	                *)
	                #PO_INVT.CTW.%B1 := 1;
	                IF "Zona".Z[#K_Zona].Gen.Reset AND ("Motore".M[#K_MotoreInt].Dati.MotoreFermo OR "Motore".M[#K_MotoreInt].In.DriverFault) THEN
	                    #PO_INVT.CTW.%B0 := 7;
	                ELSIF "Motore".M[#K_MotoreInt].Out.CmdPosMotore THEN
	                    #PO_INVT.CTW.%B0 := 1;
	                ELSIF "Motore".M[#K_MotoreInt].Out.CmdNegMotore THEN
	                    #PO_INVT.CTW.%B0 := 2;
	                ELSE
	                    #PO_INVT.CTW.%B0 := 6;
	                END_IF;
	                #PO_INVT.CTW.%X15 := NOT #PI_INVT.STW.%X15;
	                #PO_INVT.Speed := DINT_TO_INT(TRUNC("Motore".M[#K_MotoreInt].Out.VelAss / DINT_TO_REAL("Motore".M[#K_MotoreInt].Prm.C.VelMax) * 10000.0));
	                REGION ScritturaParametri
	                    IF #PI_INVT.PKW01 <> 0 THEN
	                        IF "Motore".M[#K_MotoreInt].Dati.PrmSend THEN
	                            "Motore".M[#K_MotoreInt].Dati.IdPrm += 1;
	                            IF "Motore".M[#K_MotoreInt].Dati.IdPrm > 1 THEN
	                                "Motore".M[#K_MotoreInt].Dati.IdPrm := 0;
	                            END_IF;
	                            "Motore".M[#K_MotoreInt].Dati.PrmSend := false;
	                        END_IF;
	                    ELSE
	                        "Motore".M[#K_MotoreInt].Dati.PrmSend := true;
	                        CASE "Motore".M[#K_MotoreInt].Dati.IdPrm OF
	                            0:  //Acc
	                                #PO_INVT.PKW01 := 4;
	                                #PO_INVT.PKW02 := 11;
	                                #PO_INVT.PKW04 := DINT_TO_WORD(TRUNC(DINT_TO_REAL("Motore".M[#K_MotoreInt].Prm.C.VelMax) / DINT_TO_REAL("Motore".M[#K_MotoreInt].Prm.DecEmergenza) * 3.0));
	                            1:  //Dec
	                                #PO_INVT.PKW01 := 4;
	                                #PO_INVT.PKW02 := 12;
	                                #PO_INVT.PKW04 := DINT_TO_WORD(TRUNC(DINT_TO_REAL("Motore".M[#K_MotoreInt].Prm.C.VelMax) / DINT_TO_REAL("Motore".M[#K_MotoreInt].Prm.DecEmergenza) * 3.0));
	                            ELSE
	                                "Motore".M[#K_MotoreInt].Dati.PrmSend := false;
	                                "Motore".M[#K_MotoreInt].Dati.IdPrm := 0;
	                        END_CASE;
	                    END_IF;
	                END_REGION
	                "Motore".M[#K_MotoreInt].Dati.RetVal_SCR_Inv := DPWR_DAT(LADDR := "Motore".M[#K_MotoreInt].HW.HWIO_Inverter, RECORD := #PO_INVT);
	                "Motore".M[#K_MotoreInt].HMI.CTW1 := #PO_INVT.CTW;
	            END_REGION
	        9:
	            REGION Nidec
	                (*
	                BIT 00: Drive Enable
	                BIT 01: Run Forward
	                BIT 02: Jog Forward
	                BIT 03: Run Reverse
	                BIT 04: Forward/Reverse
	                BIT 05: Run
	                BIT 06: Not Stop
	                BIT 07: Auto / manual
	                BIT 08: Analog / Preset reference
	                BIT 09: Jog Reverse
	                BIT 10: Not used
	                BIT 11: Not used
	                BIT 12: Trip drive
	                BIT 13: Reset drive
	                BIT 14: Watchdog
	                *)
	                #PO_Nidec.CTW.%X7 := true;
	                #PO_Nidec.CTW.%X0 := #PO_Nidec.CTW.%X6 := #PI_Nidec.STW.%X0 AND "Zona".Z[#K_ZonaInt].Out.CentralinaOk;
	                //#PO_Nidec.CTW.%X1 := "Motor".M[#MotorNumber].o.CmdFWD OR "Motor".M[#MotorNumber].o.CmdBKW;
	                //#PO_Nidec.CTW.%X3 := "Motor".M[#MotorNumber].o.CmdBKW;
	                #PO_Nidec.CTW.%X5 := "Motore".M[#K_MotoreInt].Out.CmdPosMotore OR "Motore".M[#K_MotoreInt].Out.CmdNegMotore;
	                #PO_Nidec.CTW.%X4 := "Motore".M[#K_MotoreInt].Out.CmdNegMotore;
	                #PO_Nidec.CTW.%X13 := "Zona".Z[#K_Zona].Gen.Reset AND "Motore".M[#K_MotoreInt].In.DriverFault;
	                #PO_Nidec.Speed := TRUNC("Motore".M[#K_MotoreInt].Out.VelAss / DINT_TO_REAL("Motore".M[#K_MotoreInt].Prm.C.VelMax) * 10000.0);
	                #PO_Nidec.RampAcc := TRUNC(DINT_TO_REAL("Motore".M[#K_MotoreInt].Prm.C.VelMax) / DINT_TO_REAL("Motore".M[#K_MotoreInt].Dati.AccRichPerc) * 3.0);
	                #PO_Nidec.RampDec := TRUNC(DINT_TO_REAL("Motore".M[#K_MotoreInt].Prm.C.VelMax) / DINT_TO_REAL("Motore".M[#K_MotoreInt].Dati.DecReqEmergInLavo) * 3.0);
	                "Motore".M[#K_MotoreInt].HMI.CTW1 := #PO_Nidec.CTW;
	                //VariantPut(SRC := #PO_Nidec, DST := #PO_Inv);
	            END_REGION
	            ;
	    END_CASE;
	END_REGION ;
	REGION Update
	    IF "Motore".M[#K_MotoreInt].HMI.UpdParam THEN
	        "Motore".M[#K_MotoreInt].HMI.UpdParam := FALSE;
	        "Motore".M[#K_MotoreInt].Out.UpdParam := true;
	    ELSE
	        IF "Motore".M[#K_MotoreInt].Out.UpdParam THEN
	            "Motore".M[#K_MotoreInt].HMI.FBGestione := 100 + "Motore".M[#K_MotoreInt].HW.TipoCollInverter;
	            CASE "Motore".M[#K_MotoreInt].HW.TipoEncoder OF
	                1: // ENCODER SICK
	                    "Motore".M[#K_MotoreInt].Dati.Encoder.RicircoloEncoder := 1073741824;
	                    "Motore".M[#K_MotoreInt].Dati.Encoder.MezzoRicircoloEncoder := "Motore".M[#K_MotoreInt].Dati.Encoder.RicircoloEncoder / 2;
	                    "Motore".M[#K_MotoreInt].Prm.Enc.ImpRev := 262144.0;
	                10, 11: // ENCODER T+R
	                    "Motore".M[#K_MotoreInt].Dati.Encoder.RicircoloEncoder := 16#0200_0000;
	                    "Motore".M[#K_MotoreInt].Dati.Encoder.MezzoRicircoloEncoder := "Motore".M[#K_MotoreInt].Dati.Encoder.RicircoloEncoder / 2;
	                    "Motore".M[#K_MotoreInt].Prm.Enc.ImpRev := 8192.0;
	            END_CASE;
	        END_IF;
	        "Motore".M[#K_MotoreInt].Out.UpdParam := false;
	    END_IF;
	    IF "Motore".M[#K_MotoreInt].Out.UpdParam THEN
	        "Motore".M[#K_MotoreInt].In.Positioning := false;
	        "Motore".M[#K_MotoreInt].In.PosRelativo := false;
	        "Motore".M[#K_MotoreInt].In.CambioVelDaPunto := false;
	        "Motore".M[#K_MotoreInt].In.CmdPosRich := false;
	        "Motore".M[#K_MotoreInt].In.CmdNegRich := false;
	        "Motore".M[#K_MotoreInt].In.MotoreRun := false;
	        "Motore".M[#K_MotoreInt].In.AttivaLimVarPos := false;
	        "Motore".M[#K_MotoreInt].In.AttivaLimVarNeg := false;
	        "Motore".M[#K_MotoreInt].In.Premagnetizza := false;
	        "Motore".M[#K_MotoreInt].In.PremagnetizzaPos := false;
	        "Motore".M[#K_MotoreInt].In.PremagnetizzaNeg := false;
	        "Motore".M[#K_MotoreInt].In.ForzaEndLessPos := false;
	        "Motore".M[#K_MotoreInt].In.ForzaEndLessNeg := false;
	        "Motore".M[#K_MotoreInt].In.ForzaEndLessBreve := false;
	        "Motore".M[#K_MotoreInt].In.SezAperto := false;
	        "Motore".M[#K_MotoreInt].In.DriverFault := false;
	        "Motore".M[#K_MotoreInt].In.DriverWarning := false;
	        "Motore".M[#K_MotoreInt].In.NoComunInv := false;
	        "Motore".M[#K_MotoreInt].In.NoComunEnc := false;
	        "Motore".M[#K_MotoreInt].In.TerVentolaOff := false;
	        "Motore".M[#K_MotoreInt].In.CinghiaRotta := false;
	        "Motore".M[#K_MotoreInt].In.SensAzz := false;
	        "Motore".M[#K_MotoreInt].In.SpinaSicNoInPos := false;
	        "Motore".M[#K_MotoreInt].In.ConsMovimentoPos := true;
	        "Motore".M[#K_MotoreInt].In.ConsMovimentoNeg := true;
	        "Motore".M[#K_MotoreInt].In.AnticadutaOFF := false;
	        "Motore".M[#K_MotoreInt].In.AnticadutaON := false;
	        "Motore".M[#K_MotoreInt].In.PercentualeRichiesta := 100;
	        "Motore".M[#K_MotoreInt].Out.CmdPosMotore := false;
	        "Motore".M[#K_MotoreInt].Out.CmdNegMotore := false;
	        "Motore".M[#K_MotoreInt].Out.CmdAnticaduta := false;
	        "Motore".M[#K_MotoreInt].Out.Paw := 0;
	        "Motore".M[#K_MotoreInt].Out.VelEncoder := 0;
	        "Motore".M[#K_MotoreInt].Prm.ByPassAnticaduta := false;
	        "Motore".M[#K_MotoreInt].Prm.AnticadutaPresente := false;
	        "Motore".M[#K_MotoreInt].Prm.PremaNoFreno := false;
	        "Motore".M[#K_MotoreInt].Prm.EscludiFunzPos := false;
	        "Motore".M[#K_MotoreInt].Prm.CambioDirNoFreno := false;
	        "Motore".M[#K_MotoreInt].Prm.CalcTempoRimanente := false;
	        "Motore".M[#K_MotoreInt].Prm.FrenoPresente := false;
	        "Motore".M[#K_MotoreInt].Prm.DisabCicloAutoAllarme := false;
	        "Motore".M[#K_MotoreInt].Prm.DisabCicloManuAllarme := false;
	        "Motore".M[#K_MotoreInt].HMI.Setup := false;
	        "Motore".M[#K_MotoreInt].HMI.ManMov := false;
	        "Motore".M[#K_MotoreInt].HMI.Param.Read := false;
	        "Motore".M[#K_MotoreInt].HMI.Param.Write := false;
	        "Motore".M[#K_MotoreInt].HMI.Param.Save := false;
	        "Motore".M[#K_MotoreInt].HMI.Param.FactoryInit := false;
	        "Motore".M[#K_MotoreInt].HMI.Param.Init_Motor := false;
	        "Motore".M[#K_MotoreInt].HMI.FBGestione := 100 + "Motore".M[#K_MotoreInt].HW.TipoCollInverter;
	        CASE "Motore".M[#K_MotoreInt].HW.TipoEncoder OF
	            1: // ENCODER SICK
	                "Motore".M[#K_MotoreInt].Dati.Encoder.RicircoloEncoder := 1073741824;
	                "Motore".M[#K_MotoreInt].Dati.Encoder.MezzoRicircoloEncoder := "Motore".M[#K_MotoreInt].Dati.Encoder.RicircoloEncoder / 2;
	                "Motore".M[#K_MotoreInt].Prm.Enc.ImpRev := 262144.0;
	            10, 11: // ENCODER T+R
	                "Motore".M[#K_MotoreInt].Dati.Encoder.RicircoloEncoder := 16#0200_0000;
	                "Motore".M[#K_MotoreInt].Dati.Encoder.MezzoRicircoloEncoder := "Motore".M[#K_MotoreInt].Dati.Encoder.RicircoloEncoder / 2;
	                "Motore".M[#K_MotoreInt].Prm.Enc.ImpRev := 8192.0;
	        END_CASE;
	        REGION CalcoloSviluppoEncoder
	            CASE "Motore".M[#K_MotoreInt].Prm.Enc.Mounting OF
	                1:
	                    // Albero Lento
	                    "Motore".M[#K_MotoreInt].Prm.C.SpazioGiroEncoder := UDINT_TO_REAL("Motore".M[#K_MotoreInt].Prm.Mech.FeedConstant);
	                2:
	                    // Albero Veloce
	                    "Motore".M[#K_MotoreInt].Prm.C.SpazioGiroEncoder := UDINT_TO_REAL("Motore".M[#K_MotoreInt].Prm.Mech.FeedConstant * "Motore".M[#K_MotoreInt].Prm.Mech.GearIn) / DINT_TO_REAL("Motore".M[#K_MotoreInt].Prm.Mech.GearOut);
	                ELSE
	                    "Motore".M[#K_MotoreInt].Prm.C.SpazioGiroEncoder := UDINT_TO_REAL("Motore".M[#K_MotoreInt].Prm.Enc.FeedConstant);
	            END_CASE;
	        END_REGION
	        "Motore".M[#K_MotoreInt].Prm.C.VelMax := TRUNC(UDINT_TO_REAL("Motore".M[#K_MotoreInt].Prm.Mech.FeedConstant) * (DINT_TO_REAL("Motore".M[#K_MotoreInt].Prm.Mech.GearIn) / DINT_TO_REAL("Motore".M[#K_MotoreInt].Prm.Mech.GearOut)) * DINT_TO_REAL("Motore".M[#K_MotoreInt].Prm.Mech.RPMMaxRef) / 60.0);
	        CASE "Motore".M[#K_MotoreInt].HMI.ModoInizializza OF
	            1:
	                "Motore".M[#K_MotoreInt].Prm.TMinVCost := 200;
	                "Motore".M[#K_MotoreInt].Prm.TCambioDir := 200;
	                IF "Motore".M[#K_MotoreInt].HW.TipoCollInverter <> 0 THEN
	                    "Motore".M[#K_MotoreInt].Prm.VelPrema := 1;
	                ELSE
	                    "Motore".M[#K_MotoreInt].Prm.VelPrema := "Motore".M[#K_MotoreInt].Prm.C.VelMax / 100;
	                END_IF;
	                "Motore".M[#K_MotoreInt].Prm.VelBassa := "Motore".M[#K_MotoreInt].Prm.C.VelMax / 10;
	                "Motore".M[#K_MotoreInt].Prm.VelSgancioFrenoPos := "Motore".M[#K_MotoreInt].Prm.C.VelMax / 50;
	                "Motore".M[#K_MotoreInt].Prm.VelSgancioFrenoNeg := "Motore".M[#K_MotoreInt].Prm.C.VelMax / 50;
	                "Motore".M[#K_MotoreInt].Prm.SpazioArrestoPos := "Motore".M[#K_MotoreInt].Prm.C.VelMax / 500;
	                "Motore".M[#K_MotoreInt].Prm.SpazioArrestoNeg := "Motore".M[#K_MotoreInt].Prm.C.VelMax / 500;
	                "Motore".M[#K_MotoreInt].Prm.Precisione := MAX(IN1 := "Motore".M[#K_MotoreInt].Prm.SpazioArrestoPos, IN2 := "Motore".M[#K_MotoreInt].Prm.SpazioArrestoNeg) * 2;
	                "Motore".M[#K_MotoreInt].Prm.Inerzia := "Motore".M[#K_MotoreInt].Prm.Precisione + 2000;
	                "Motore".M[#K_MotoreInt].Prm.DecFinale := "Motore".M[#K_MotoreInt].Prm.C.VelMax * 2;
	                "Motore".M[#K_MotoreInt].Prm.DecEmergenza := "Motore".M[#K_MotoreInt].Prm.C.VelMax * 3;
	                "Motore".M[#K_MotoreInt].In.Acc := "Motore".M[#K_MotoreInt].Prm.C.VelMax * 2;
	                "Motore".M[#K_MotoreInt].In.Dec := "Motore".M[#K_MotoreInt].Prm.C.VelMax * 2;
	                "Motore".M[#K_MotoreInt].Prm.VelMan := "Motore".M[#K_MotoreInt].Prm.C.VelMax / 4;
	                "Motore".M[#K_MotoreInt].Prm.VelJog := "Motore".M[#K_MotoreInt].Prm.C.VelMax / 10;
	                "Motore".M[#K_MotoreInt].Prm.ValMaxRef := 27648;
	            2:
	                "Motore".M[#K_MotoreInt].Prm.TMinVCost := 200;
	                "Motore".M[#K_MotoreInt].Prm.TCambioDir := 200;
	                IF "Motore".M[#K_MotoreInt].HW.TipoCollInverter <> 0 THEN
	                    "Motore".M[#K_MotoreInt].Prm.VelPrema := 1;
	                ELSE
	                    "Motore".M[#K_MotoreInt].Prm.VelPrema := "Motore".M[#K_MotoreInt].Prm.C.VelMax / 100;
	                END_IF;
	                "Motore".M[#K_MotoreInt].Prm.VelBassa := "Motore".M[#K_MotoreInt].Prm.C.VelMax / 10;
	                "Motore".M[#K_MotoreInt].Prm.VelSgancioFrenoPos := "Motore".M[#K_MotoreInt].Prm.C.VelMax / 25;
	                "Motore".M[#K_MotoreInt].Prm.VelSgancioFrenoNeg := "Motore".M[#K_MotoreInt].Prm.C.VelMax / 25;
	                "Motore".M[#K_MotoreInt].Prm.SpazioArrestoPos := "Motore".M[#K_MotoreInt].Prm.C.VelMax / 500;
	                "Motore".M[#K_MotoreInt].Prm.SpazioArrestoNeg := "Motore".M[#K_MotoreInt].Prm.C.VelMax / 500;
	                "Motore".M[#K_MotoreInt].Prm.Precisione := MAX(IN1 := "Motore".M[#K_MotoreInt].Prm.SpazioArrestoPos, IN2 := "Motore".M[#K_MotoreInt].Prm.SpazioArrestoNeg) * 2;
	                "Motore".M[#K_MotoreInt].Prm.Inerzia := "Motore".M[#K_MotoreInt].Prm.Precisione + 2000;
	                "Motore".M[#K_MotoreInt].Prm.DecFinale := "Motore".M[#K_MotoreInt].Prm.C.VelMax * 2;
	                "Motore".M[#K_MotoreInt].Prm.DecEmergenza := "Motore".M[#K_MotoreInt].Prm.C.VelMax * 3;
	                "Motore".M[#K_MotoreInt].In.Acc := "Motore".M[#K_MotoreInt].Prm.C.VelMax * 2;
	                "Motore".M[#K_MotoreInt].In.Dec := "Motore".M[#K_MotoreInt].Prm.C.VelMax * 2;
	                "Motore".M[#K_MotoreInt].Prm.VelMan := "Motore".M[#K_MotoreInt].Prm.C.VelMax / 4;
	                "Motore".M[#K_MotoreInt].Prm.VelJog := "Motore".M[#K_MotoreInt].Prm.C.VelMax / 10;
	                "Motore".M[#K_MotoreInt].Prm.ValMaxRef := 27648;
	            3:
	                "Motore".M[#K_MotoreInt].Prm.TMinVCost := 200;
	                "Motore".M[#K_MotoreInt].Prm.TCambioDir := 200;
	                IF "Motore".M[#K_MotoreInt].HW.TipoCollInverter <> 0 THEN
	                    "Motore".M[#K_MotoreInt].Prm.VelPrema := 1;
	                ELSE
	                    "Motore".M[#K_MotoreInt].Prm.VelPrema := "Motore".M[#K_MotoreInt].Prm.C.VelMax / 100;
	                END_IF;
	                "Motore".M[#K_MotoreInt].Prm.VelBassa := "Motore".M[#K_MotoreInt].Prm.C.VelMax / 10;
	                "Motore".M[#K_MotoreInt].Prm.VelSgancioFrenoPos := "Motore".M[#K_MotoreInt].Prm.C.VelMax / 25;
	                "Motore".M[#K_MotoreInt].Prm.VelSgancioFrenoNeg := "Motore".M[#K_MotoreInt].Prm.C.VelMax / 25;
	                "Motore".M[#K_MotoreInt].Prm.SpazioArrestoPos := "Motore".M[#K_MotoreInt].Prm.C.VelMax / 500;
	                "Motore".M[#K_MotoreInt].Prm.SpazioArrestoNeg := "Motore".M[#K_MotoreInt].Prm.C.VelMax / 500;
	                "Motore".M[#K_MotoreInt].Prm.Precisione := MAX(IN1 := "Motore".M[#K_MotoreInt].Prm.SpazioArrestoPos, IN2 := "Motore".M[#K_MotoreInt].Prm.SpazioArrestoNeg) * 2;
	                "Motore".M[#K_MotoreInt].Prm.Inerzia := "Motore".M[#K_MotoreInt].Prm.Precisione + 2000;
	                "Motore".M[#K_MotoreInt].Prm.DecFinale := "Motore".M[#K_MotoreInt].Prm.C.VelMax;
	                "Motore".M[#K_MotoreInt].Prm.DecEmergenza := "Motore".M[#K_MotoreInt].Prm.C.VelMax;
	                "Motore".M[#K_MotoreInt].In.Acc := "Motore".M[#K_MotoreInt].Prm.C.VelMax / 2;
	                "Motore".M[#K_MotoreInt].In.Dec := "Motore".M[#K_MotoreInt].Prm.C.VelMax / 2;
	                "Motore".M[#K_MotoreInt].Prm.VelMan := "Motore".M[#K_MotoreInt].Prm.C.VelMax / 4;
	                "Motore".M[#K_MotoreInt].Prm.VelJog := "Motore".M[#K_MotoreInt].Prm.C.VelMax / 10;
	                "Motore".M[#K_MotoreInt].Prm.ValMaxRef := 27648;
	        END_CASE;
	        "Motore".M[#K_MotoreInt].HMI.ModoInizializza := 0;
	        "Motore".M[#K_MotoreInt].Allarmi.WordHmi_1 :=
	        "Motore".M[#K_MotoreInt].Allarmi.WordHmi_2 := 0;
	    END_IF;
	END_REGION ;
	REGION Motor block
	    IF "Motore".M[#K_MotoreInt].Dati.MotorStop THEN
	        IF NOT "Motore".M[#K_MotoreInt].Out.InMarcia THEN
	            IF "Motore".M[#K_MotoreInt].Dati.AlmInv_RitRestart > 1000 THEN
	                "Motore".M[#K_MotoreInt].Dati.MotorStop := false;
	            ELSE
	                "Motore".M[#K_MotoreInt].Dati.AlmInv_RitRestart += REAL_TO_INT("Zona".Comuni.TempoCicloCpu_r);
	            END_IF;
	        ELSE
	            "Motore".M[#K_MotoreInt].Dati.AlmInv_RitRestart := 0;
	        END_IF;
	    END_IF;
	    IF "Motore".M[#K_MotoreInt].Dati.AlmBloccato_Cont > 0 OR"Motore".M[#K_MotoreInt].Dati.AlmInv_Cont > 0 THEN
	        "Motore".M[#K_MotoreInt].Dati.Alm_ContAzzCont += REAL_TO_INT("Zona".Comuni.TempoCicloCpu_r);
	        IF "Motore".M[#K_MotoreInt].Dati.Alm_ContAzzCont > 60000 THEN
	            "Motore".M[#K_MotoreInt].Dati.AlmBloccato_Cont := 0;
	            "Motore".M[#K_MotoreInt].Dati.AlmInv_Cont := 0;
	            "Motore".M[#K_MotoreInt].Dati.Alm_ContAzzCont := 0;
	        END_IF;
	    ELSE
	        "Motore".M[#K_MotoreInt].Dati.Alm_ContAzzCont := 0;
	    END_IF;
	END_REGION ;
	REGION Riferimenti incrociati
	    "Motore".M[#K_MotoreInt].Rif_Inc.K_Analogica := "Motore".M[#K_MotoreInt].Prm.K_Analogica;
	    "Motore".M[#K_MotoreInt].Rif_Inc.K_Zona := #K_ZonaInt;
	END_REGION ;
	REGION Pulisco i comandi della sequenza
	    IF "Motore".M[#K_MotoreInt].Dati.InclusoInUnaSequenza THEN
	        "Motore".M[#K_MotoreInt].In.CmdPosRich :=
	        "Motore".M[#K_MotoreInt].In.CmdNegRich := False;
	    END_IF;
	END_REGION ;
END_FUNCTION

